Fanuc KAREL source: ka00040.KL

PROGRAM KA00040
%NOLOCKGROUP
VAR
SRC : STRING[80];DST : STRING[80]
BEGIN
--
SRC='A'
DST=SRC
END KA00040
